ABB RobotStudio station: ProjetoDomino.rsstn

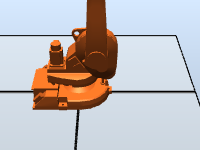
Station ProjetoDomino (saved by RobotStudio 6.8.8148.134)
Controller IRB_1600_6kg_1.45m
  mechanical unit ROB_1: IRB1600_5_145__01, 6 joints, base frame (0, 0, 0) mm
Layout (positions relative to the parent item):
  - IRB1600_5_145__01 [mechanism, from Robots\IRB1600_5_145__01.rslib] at (0, 0, 0) mm; joint values [0, 0, 0, 0, 0.5236, 0] (rad or m)
